FUNCTION_BLOCK Infeed EXTENDS FB_PackML_BaseModule
VAR
END_VAR

// This method serves as the entry point for all underlying FB logic
METHOD PUBLIC CyclicLogic

// This method should be called cyclically by descendant function blocks by invoking SUPER^.CyclicLogic().  Alternatively, the contents of this method could be reimplemented entirely in which case a call to this method would not be necessary.
IF NOT _InitComplete THEN
	_InitComplete := Initialize();
	RETURN;
END_IF

SUPER^.CyclicLogic();
END_METHOD

// Basic module initialization logic
METHOD PROTECTED Initialize : BOOL;

// This method is called by CyclicLogic() as required
Initialize := FALSE;
CASE DescendantSequenceState OF
	0:
		//Setup Config
		_LogModeChanges			:= FALSE;
		_LogStateChanges		:= FALSE;
		DescendantSequenceState := DescendantSequenceState + 10;

	10: // Call the Super to Initialize all SubModules and Components
		IF SUPER^.Initialize() THEN
			Initialize := TRUE;
		END_IF
END_CASE
END_METHOD

END_FUNCTION_BLOCK

(* stored: Version 1.1.0.1, ProductVersion 3.1.4026.13
   POU Infeed: Id {76aab0a3-2381-4d9d-a825-dafde1ec23bf}, SpecialFunc None
   Method CyclicLogic: Id {b56ad18f-453b-4183-a853-5b8d97a37ec6}
   Method Initialize: Id {9c852996-617e-486f-b4eb-534d46aa5a77} *)
